SUBAPPLICATION GreenWhiteBackground4_AXC (* Hintergrundfarbe (TRUE -> Grün, FALSE -> Weiß) für 4 Objekte (AX-Adapter) (Kompakt) *)
  (* Standard: 61499-2 *)
  (* Version 1.0, 2026-07-21, franz, Meisterschulen am Ostbahnhof *)
  PACKAGE MyLib::sys;
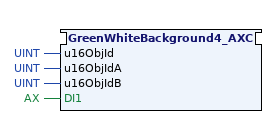
  VAR_INPUT
    u16ObjId : UINT;
    u16ObjIdA : UINT;
    u16ObjIdB : UINT;
  END_VAR
  SOCKETS
    DI1 : adapter::types::unidirectional::AX;
  END_SOCKETS
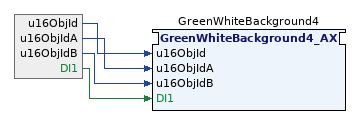
  SUBAPPS
    GreenWhiteBackground4 : MyLib::sys::GreenWhiteBackground4_AX;
  END_SUBAPPS
  DATA_CONNECTIONS
    u16ObjId TO GreenWhiteBackground4.u16ObjId;
    u16ObjIdA TO GreenWhiteBackground4.u16ObjIdA;
    u16ObjIdB TO GreenWhiteBackground4.u16ObjIdB;
  END_CONNECTIONS
  ADAPTER_CONNECTIONS
    DI1 TO GreenWhiteBackground4.DI1;
  END_CONNECTIONS
END_SUBAPPLICATION
